(* IEC 61131-3 sources: Studia/Automatyka BR/Suwnica/Soft/Code/Program, 2 files *)

(* ---- Types.typ ---- *)
TYPE
(*	OperatorTyp : STRUCT
		diStart : BOOL;
		diStop : BOOL;
		diReset : BOOL;
		doAktywny : BOOL;
		doPrawo : BOOL;
		doLewo : BOOL;
	END_STRUCT;*)

	GateTyp : STRUCT
		diOtwarte : BOOL;
		diZamkniete : BOOL;
		doZasilanie : BOOL;
		doPrawoLewo : BOOL;
		doLampa : BOOL;
		uiOtwarte : BOOL;
		uiZamkniete : BOOL;
		uiZasilanie : BOOL;
		uiPrawoLewo : BOOL;
		uiLampa : BOOL;
		Pilot : PilotTyp;
		diKrancowkaLewo : BOOL;
		diKrancowkaPrawo : BOOL;
		SilnikDC : SilnikDCTyp;
	END_STRUCT;

	SilnikDCTyp : STRUCT
		aoPWM : INT;
		PeriodDuration : UINT;
	END_STRUCT;

	EnkoderABTyp : STRUCT (*enkoder do suwnicy, jak chcemy np przeskalowac pozycje na milimetry*)
		aiPozycja : DINT;
		uiPozycja : REAL;
		uiTryb : USINT; (**ustawić na 195*)
	END_STRUCT;

	PilotTyp : STRUCT
		diOtworz : BOOL;
		diZamknij : BOOL;
		doStanBramy : BOOL;
		uiOtwieranie : BOOL;
		uiZamykanie : BOOL;
		aiZadajnik : ARRAY[1..2] OF INT;
	END_STRUCT;

	HouseTyp : STRUCT
		Brama : GateTyp;
	END_STRUCT;

	StatemachineTyp:
		(
		WAIT_FOR_ACTION :=1,
		HOMING :=2,
		GO_TO_START :=3,
		WAIT_FOR_ITEM :=4,
		GO_TO_END :=5,
		WAIT_FOR_OUT :=6,
		FAILURE :=7,
		GO_TO_START0:=8
	);

	SuwnicaTyp : STRUCT
		diStartLS_NC : BOOL;
		diStartLS_NO : BOOL;
		diEndLS_NC : BOOL;
		diEndLS_NO : BOOL;
		diItemStart : BOOL;
		diItemEnd : BOOL;
		SilnikDC : SilnikDCTyp;
		Enkoder : EnkoderABTyp;
		Operator : OperatorTyp;
	(*	aiPozycja : DINT; *)
	END_STRUCT;

	OperatorTyp :STRUCT
		diStart : BOOL;
		diStop : BOOL;
		diESTOP : BOOL;
		diReset : BOOL;
		doAktywny : BOOL;
		doAwaria : BOOL;

	END_STRUCT;

	SuwnicaParTyp : STRUCT
		uiHomingSpeed : INT;
		uiGoToStartSpeed: ARRAY[1..2] OF UINT;
		uiGoToEndSpeed : INT;
		uiStartPozycja : ARRAY[1..2] OF DINT;
		uiEndPozycja : ARRAY[1..2] OF DINT;
		uiTolPozycja : DINT;

	END_STRUCT;
END_TYPE

(* ---- Main.st ---- *)
PROGRAM _INIT
	ControlTyp:=5;
	Suwnica.SilnikDC.PeriodDuration:=100;
	Maszynastanu:=WAIT_FOR_ACTION;
	Suwnica.Enkoder.uiTryb:=195;
END_PROGRAM

PROGRAM _CYCLIC
	CASE ControlTyp OF
		1: //sterowanie logicyne
			Dom.Brama.doZasilanie:=Dom.Brama.Pilot.diOtworz XOR Dom.Brama.Pilot.diZamknij;
			Dom.Brama.doPrawoLewo:=Dom.Brama.Pilot.diOtworz AND NOT Dom.Brama.Pilot.diZamknij;

		2:
			Dom.Brama.doZasilanie:=Dom.Brama.Pilot.uiOtwieranie XOR Dom.Brama.Pilot.uiZamykanie;
			Dom.Brama.doPrawoLewo:=Dom.Brama.Pilot.uiOtwieranie AND NOT Dom.Brama.Pilot.uiZamykanie;

			temp1:=Dom.Brama.Pilot.uiOtwieranie;

			Dom.Brama.Pilot.uiOtwieranie:=(EDGEPOS(Dom.Brama.Pilot.diOtworz) OR Dom.Brama.Pilot.uiOtwieranie) AND NOT(Dom.Brama.Pilot.diZamknij OR Dom.Brama.Pilot.uiZamykanie OR Dom.Brama.diKrancowkaPrawo); // operacja zapisu do pamięci
			Dom.Brama.Pilot.uiZamykanie:=(EDGEPOS(Dom.Brama.Pilot.diZamknij) OR Dom.Brama.Pilot.uiZamykanie) AND NOT(Dom.Brama.Pilot.diOtworz OR temp1 OR Dom.Brama.diKrancowkaLewo);

		4:
			Skaluj[1].x:=INT_TO_REAL(Dom.Brama.Pilot.aiZadajnik[1]);
			Skaluj[1].x1:=0;
			Skaluj[1].y1:=-32768;
			Skaluj[1].x2:=32767;
			Skaluj[1].y2:=32767;
			Skaluj[1]();
			Suwnica.SilnikDC.aoPWM:=REAL_TO_INT(Skaluj[1].y);
			IF EDGEPOS(Suwnica.diStartLS_NC)=TRUE OR EDGEPOS(Suwnica.diEndLS_NC)=TRUE THEN
				Suwnica.SilnikDC.aoPWM:=0;

			END_IF;

		5:
			(*IF fLoadDefaults THEN
				SuwnicaPar.uiTolPoyzcja:=1000;
				SuwnicaPar.uiHomingSpeed:=2000;
				SuwnicaPar.uiGoToStartSpeed:=
				SuwnicaPar.uiGoToEndSpeed := -15000;
				SuwnicaPar.uiStartPozycja[1] :=14000;
				SuwnicaPar.uiEndPozycja :=
				SuwnicaPar.uiTolPozycja :=

				uipositionstart1 14000
				uiendposition1 90000
				homingspeed 2000
				gotostartspeed1 -5000
				gotostartspeed2 5000
				gotoendspeed1 -15000*)

			CASE Maszynastanu OF
				WAIT_FOR_ACTION:
					IF Suwnica.Operator.diStart AND (Suwnica.Enkoder.aiPozycja <= 100) AND (Suwnica.Enkoder.aiPozycja >= -100) AND Suwnica.diStartLS_NC THEN
						Maszynastanu:=GO_TO_START;

					END_IF;

					IF Suwnica.Operator.diStart AND ((Suwnica.Enkoder.aiPozycja > 100) OR (Suwnica.Enkoder.aiPozycja < -100) OR Suwnica.diStartLS_NC = FALSE)  THEN
						Maszynastanu:=HOMING;

					END_IF;

				HOMING:
					Suwnica.SilnikDC.aoPWM:= 12000;
					IF EDGEPOS(Suwnica.diEndLS_NC)=TRUE THEN
						Suwnica.SilnikDC.aoPWM:= 0;
						Maszynastanu:= GO_TO_START0;

					END_IF;
				GO_TO_START0:
					Suwnica.SilnikDC.aoPWM:= -16000;
					IF (Suwnica.Enkoder.aiPozycja <= 42000) AND (Suwnica.Enkoder.aiPozycja >=38000) THEN
						Suwnica.SilnikDC.aoPWM:= 0;
						Maszynastanu:= WAIT_FOR_ITEM;
					END_IF;

					IF Suwnica.Operator.diStop OR Suwnica.Operator.diESTOP THEN
						Suwnica.SilnikDC.aoPWM:= 0;
						Maszynastanu:=WAIT_FOR_ACTION;
					END_IF;

				GO_TO_START:
					Suwnica.SilnikDC.aoPWM:= 16000;
					IF (Suwnica.Enkoder.aiPozycja <= 42000) AND (Suwnica.Enkoder.aiPozycja >=38000) THEN
						Suwnica.SilnikDC.aoPWM:= 0;
						Maszynastanu:= WAIT_FOR_ITEM;
					END_IF;

					IF Suwnica.Operator.diStop OR Suwnica.Operator.diESTOP THEN
						Suwnica.SilnikDC.aoPWM:= 0;
						Maszynastanu:=WAIT_FOR_ACTION;
					END_IF;

				WAIT_FOR_ITEM:
					(*IF Suwnica.Operator.diStop OR Suwnica.Operator.diESTOP THEN
						Suwnica.SilnikDC.aoPWM:= 0;
						Maszynastanu:=WAIT_FOR_ACTION;*)
					//DelayON[1].IN:=Suwnica.diEndLS_NO;
					DelayON[1].IN:=Suwnica.diStartLS_NO;
					DelayON[1].PT:=T#2s;
					DelayON[1]();
					IF DelayON[1].Q THEN
						DelayON[1].IN:=FALSE;
						DelayON[1]();
						Maszynastanu:=GO_TO_END;
					END_IF;

				GO_TO_END:
					Suwnica.SilnikDC.aoPWM:= -16000;
					IF (Suwnica.Enkoder.aiPozycja <= 282000) AND (Suwnica.Enkoder.aiPozycja >=278000) THEN
						Suwnica.SilnikDC.aoPWM:= 0;

						IF NOT(Suwnica.diEndLS_NO) THEN
							Maszynastanu:=FAILURE;
						ELSE
							Maszynastanu:= WAIT_FOR_OUT;
						END_IF;

					END_IF;

					IF Suwnica.Operator.diStop OR Suwnica.Operator.diESTOP THEN
						Suwnica.SilnikDC.aoPWM:= 0;
						Maszynastanu:=WAIT_FOR_ACTION;
					END_IF;

				WAIT_FOR_OUT:

					DelayON[2].IN:=NOT(Suwnica.diEndLS_NO);
					DelayON[2].PT:=T#2s;
					DelayON[2]();
					IF DelayON[2].Q THEN
						DelayON[2].IN:=FALSE;
						DelayON[2]();
						Maszynastanu:=GO_TO_START;

					END_IF;

					FAILURE:
					Suwnica.SilnikDC.aoPWM:= 0;
					DelayON[3].IN:=NOT DelayON[3].Q;
					DelayON[3].PT:=T#300ms;
					DelayON[3]();
					Suwnica.Operator.doAwaria:=Suwnica.Operator.doAwaria XOR DelayON[3].Q;

					IF Suwnica.Operator.diReset THEN
						Suwnica.Operator.doAwaria:=FALSE;
						Maszynastanu:=WAIT_FOR_ACTION;
		 			END_IF;

			END_CASE;

	END_CASE;

END_PROGRAM

PROGRAM _EXIT

END_PROGRAM
